(* IEC 61131-3 sources: plc_generation_empirical_study/datasets/task_bank_v0_2/tasks/C01_B06_composite/negative_control, 1 file *)

(* ---- NC1.st ---- *)
FUNCTION_BLOCK C01_B06_composite
VAR_INPUT
    A_ChA : BOOL;
    A_ChB : BOOL;
    A_TestMode : BOOL;
    A_TestPermit : BOOL;
    A_ProcessRequest : BOOL;
    B_S1 : BOOL;
    B_S2 : BOOL;
    B_S3 : BOOL;
    SubsystemBEnable : BOOL;
    CrossReset : BOOL;
END_VAR
VAR_OUTPUT
    A_SafeEnable : BOOL;
    A_Disagree : BOOL;
    A_TestActive : BOOL;
    B_Vote : BOOL;
    B_Unanimous : BOOL;
    CrossReady : BOOL;
    CrossBlocked : BOOL;
END_VAR

A_Disagree := A_ChA <> A_ChB;
A_TestActive := A_TestMode AND A_TestPermit;
IF A_TestMode THEN
    A_SafeEnable := A_ProcessRequest AND A_TestPermit AND A_ChA;
ELSE
    A_SafeEnable := A_ProcessRequest AND A_ChA AND A_ChB;
END_IF;

IF CrossReset THEN
    CrossReady := FALSE;
ELSIF A_SafeEnable THEN
    CrossReady := FALSE;
END_IF;
CrossBlocked := SubsystemBEnable AND (NOT CrossReady);

IF SubsystemBEnable AND CrossReady THEN
    B_Vote := (B_S1 AND B_S2) OR (B_S1 AND B_S3) OR (B_S2 AND B_S3);
    B_Unanimous := (B_S1 AND B_S2 AND B_S3) OR ((NOT B_S1) AND (NOT B_S2) AND (NOT B_S3));
ELSE
    B_Vote := FALSE;
    B_Unanimous := FALSE;
END_IF;

END_FUNCTION_BLOCK
